INTERFACE I_GantryPallet

PROPERTY PalletReady : BOOL
GET
END_GET
END_PROPERTY

END_INTERFACE

(* stored: Version 1.1.0.1, ProductVersion 3.1.4024.4
   Itf I_GantryPallet: Id {6444b687-f8da-4df8-a3c2-de42761437ff}
   Property PalletReady: Id {cb390074-6916-4864-a02e-789f49a16aca}
   Get Get: Id {ed64a652-d2e7-4211-819d-6ca1d61eb595} *)
